FUNCTION_BLOCK ModbusReadWord EXTENDS ModbusIo
VAR_INPUT
	Override: BOOL;
	OverrideValue: INT;
END_VAR
VAR_OUTPUT
	Value: INT;
	ValueW: WORD;
END_VAR
VAR
END_VAR
VAR PERSISTENT
END_VAR

SUPER^();
IF Override THEN
	Value := OverrideValue;
END_IF
ValueW := ValueWord;

PROPERTY ValueWord : WORD
GET
IF NOT Override THEN
	ValueWord := INT_TO_WORD(Value);
ELSE
	ValueWord := INT_TO_WORD(OverrideValue);
END_IF
END_GET
SET
IF NOT Override THEN
	Value := WORD_TO_INT(ValueWord);
ELSE
	Value := OverrideValue;
END_IF
END_SET
END_PROPERTY

END_FUNCTION_BLOCK

(* stored: Version 1.1.0.1, ProductVersion 3.1.4024.6
   POU ModbusReadWord: Id {6f7dd8cb-9c2a-4cd0-91a0-b01f02154bdf}, SpecialFunc None
   Property ValueWord: Id {0242e1c3-ab32-41c2-87b7-98b4c4f1f701}
   Get Get: Id {c18f4f2a-0704-40d4-8c2b-736bf24d9821}
   Set Set: Id {b42f12fd-f678-4055-8508-90b4b8bbd69c} *)
